// TIA Portal V20 export
DATA_BLOCK "BK10"   // DB236
// stored: MemoryReserve 100
   VAR
      "X10-1 SIDE TAPE Attachment LEFT BACKWARD" : Bool;
      "X11-1 SIDE TAPE Attachment RIGHT BACKWARD" : Bool;
      "X12-1 SIDE TAPE Attachment 1 TOP VACCUM PRESSURE SWITCH" : Bool;
      "X13-1 SIDE TAPE Attachment 2 TOP VACCUM PRESSURE SWITCH" : Bool;
      "X14-1 SIDE TAPE ATTACHEMNT LEFT PRESSURE SWITCH" : Bool;
      "X15-1 SIDE TAPE Attachment BTM BACKWARD" : Bool;
      "X16-1 SIDE TAPING Y-AYIS LIMIT SENSOR(-)" : Bool;
      "X17-1 SIDE TAPING Y-AYIS LIMIT SENSOR(+)" : Bool;
      "X10-2 SIDE TAPE Attachment LEFT FORWARD" : Bool;
      "X11-2 SIDE TAPE Attachment RIGHT FORWARD" : Bool;
      "X12-2 SIDE TAPE Attachment 1 BTM VACCUM PRESSURE SWITCH" : Bool;
      "X13-2 SIDE TAPE Attachment 2 BTM VACCUM PRESSURE SWITCH" : Bool;
      "X14-2 SIDE TAPE ATTACHMENT RIGHT PRESSURE SWITCH" : Bool;
      "X15-2 SIDE TAPE Attachment BTM FORWARD" : Bool;
      "X16-2 SIDE TAPING Y-AYIS HOME SENSOR" : Bool;
      "X17-2 SPARE" : Bool;
   END_VAR
BEGIN
END_DATA_BLOCK
